ABB RobotStudio station: first_asignm.rspag

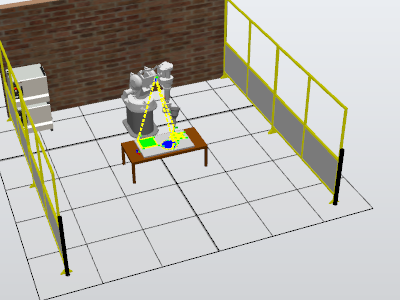
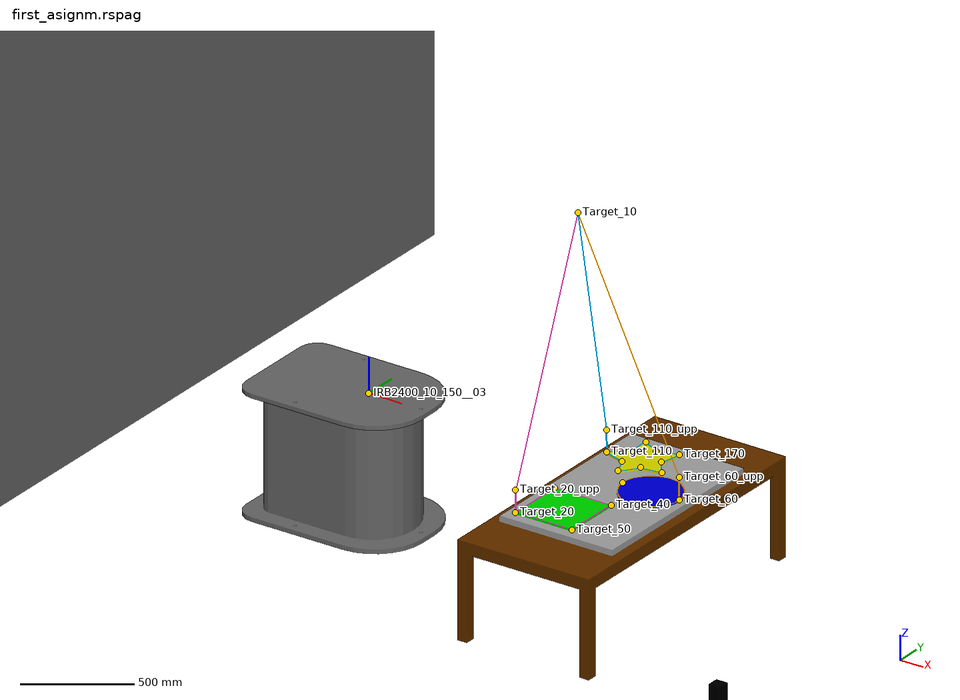
[picture v1: parts stored in the station drawn from their meshes, with robot base, taught points and paths (robot models come from the ABB library and are not in the file)]
--- station ---
Station first_asignm (saved by RobotStudio 24.1.10713.1)
Controller Controller2, task T_ROB1: task frame (RAPID world) sits at (2.56, -1.45, 620) mm, rotated rx 0 ry 0 rz -0.59 deg in the station
Controller Controller2
  mechanical unit ROB_1: IRB2400_10_150__03, 6 joints, base frame (0, 0, 0) mm
Layout (positions relative to the parent item):
  - IRB2400_10_150__03 [mechanism, from %ABB.RobotStudio.Models.IRB2400%\IRB2400_10_150_G_03.rslib] at (2.56, -1.45, 620) mm, rotated rx 0 ry 0 rz -0.59 deg; joint values [0.3771, 1.0223, 1.6235, 0.1721, -1.1317, 0.4182] (rad or m)
  - RobotStand2400H620 [part] at (0, 0, 0) mm, rotated rx 0 ry 0 rz -90 deg, size 600 x 830 x 620 mm
  - Table [part] at (1700, -750, 0) mm, rotated rx 0 ry 0 rz 90 deg, size 1500 x 700 x 488 mm
  - BackgroundWall [part] at (-1400, 2500, 0) mm, rotated rx 0 ry -90 rz 90 deg, size 2500 x 200 x 5000 mm
  - Fence_2500 [graphiccomponentgroup, from Equipment\Fence_2500.rslib] at (-1373.2, 2448.38, 0) mm, rotated rx 0 ry 0 rz -90 deg
    - Body 1 [part, from Equipment\Fence_2500.rslib]
    - Body 2 [part, from Equipment\Fence_2500.rslib]
  - Fence_2500_2 [graphiccomponentgroup, from Equipment\Fence_2500.rslib] at (1125.76, 2439.94, 0) mm, rotated rx 0 ry 0 rz -90 deg
    - Body 1 [part, from Equipment\Fence_2500.rslib]
    - Body 2 [part, from Equipment\Fence_2500.rslib]
  - Fence_2500_3 [graphiccomponentgroup, from Equipment\Fence_2500.rslib] at (-1386.44, -2458.41, 0) mm, rotated rx 0 ry 0 rz -90 deg
    - Body 1 [part, from Equipment\Fence_2500.rslib]
    - Body 2 [part, from Equipment\Fence_2500.rslib]
  - Fence_2500_4 [graphiccomponentgroup, from Equipment\Fence_2500.rslib] at (1081.61, -2474.76, 0) mm, rotated rx 0 ry 0 rz -90 deg
    - Body 1 [part, from Equipment\Fence_2500.rslib]
    - Body 2 [part, from Equipment\Fence_2500.rslib]
  - LightSensor [part] at (3608.83, 2403.41, 0) mm, size 60 x 60 x 1200 mm
  - LightSensor_2 [part] at (3563.84, -2499.97, 0) mm, size 60 x 60 x 1200 mm
  - supportframe2 [part] at (1050, 500, 488) mm, rotated rx 0 ry 0 rz -90 deg, size 1000 x 600 x 30 mm
  - star [part] at (1001.14, 175.39, 469.61) mm, rotated rx 0 ry 0 rz -18 deg, size 309.3 x 312.1 x 30 mm
  - cirkel [part] at (1023.03, -355.65, 518) mm, size 300 x 298.4 x 30 mm
  - kvadrat [part] at (460, -520, 516.18) mm, size 300 x 300 x 30 mm
  - gluetool [mechanism, from Assiment\gluetool.rslib] at (819.78, 298.44, 801.45) mm, rotated rx 143.42 ry 54.04 rz 148.38 deg
  - IRC5_Dual-Cabinet [part, from %ABB.RobotStudio.Models.IRC5%\IRC5_Dual-Cabinet.rslib] at (-784.69, -2074.47, 100) mm, rotated rx 90 ry 0 rz 90 deg
  - Part_2 [part] at (1023.03, -355.65, 518) mm, size 300 x 298.4 x 0 mm
Attachment: star is attached to supportframe2
Attachment: kvadrat is attached to supportframe2
Attachment: cirkel is attached to supportframe2
Attachment: supportframe2 is attached to Table
Attachment: gluetool is attached to IRB2400_10_150__03 / Link6

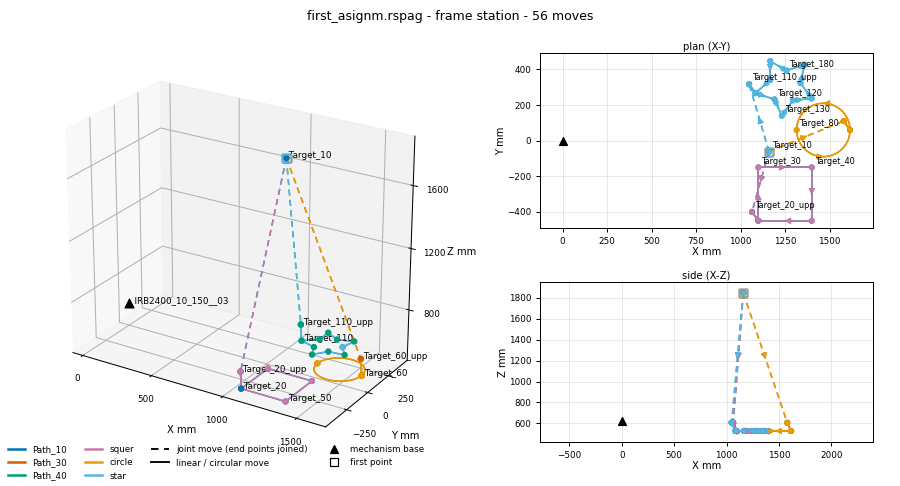
[picture p0: tool path of first_asignm.rspag in frame station, 56 of 56 moves have a stored position in this frame; points joined in program order, loops and branches not executed]
--- Backups/Controller2/RAPID/TASK1/PROGMOD/CalibData.mod ---
MODULE CalibData
    PERS tooldata gluetool:=[TRUE,[[47.792,-47.793,292.208],[0.923880453,0.270593988,0.27059897,0.000004062]],[1,[0,0,1],[1,0,0,0],0,0,0]];
    TASK PERS wobjdata Workobject_1:=[FALSE,TRUE,"",[[1465.9377766,-555.559495537,-110.643721572],[0.981995154,0.007735876,-0.020435156,0.187638159]],[[0,0,0],[1,0,0,0]]];
ENDMODULE

--- Backups/Controller2/RAPID/TASK1/PROGMOD/Module1.mod ---
MODULE Module1
        CONST robtarget Target_10:=[[-41.760657856,595.661836036,1334.239977499],[0.1634513,0.3686913,0.914955019,-0.014412176],[0,-1,0,0],[9E+09,9E+09,9E+09,9E+09,9E+09,9E+09]];
    CONST robtarget Target_20:=[[-293.739133821,244.320639444,27.648533238],[0.164058227,0.357731456,0.916814008,-0.067566099],[0,-1,0,0],[9E+09,9E+09,9E+09,9E+09,9E+09,9E+09]];
    CONST robtarget Target_30:=[[-186.145059876,524.28142208,20.904985353],[0.164039379,0.358304337,0.91678529,-0.064913921],[0,-1,0,0],[9E+09,9E+09,9E+09,9E+09,9E+09,9E+09]];
    CONST robtarget Target_40:=[[93.599135006,416.499861723,9.665738199],[0.163835348,0.362975372,0.916283469,-0.042795602],[0,-1,0,0],[9E+09,9E+09,9E+09,9E+09,9E+09,9E+09]];
    CONST robtarget Target_50:=[[-13.994938939,136.539079087,16.409286084],[0.164008319,0.359172644,0.916728515,-0.060869634],[0,-1,0,0],[9E+09,9E+09,9E+09,9E+09,9E+09,9E+09]];
    CONST robtarget Target_60:=[[369.476992779,535.242345722,-1.285956973],[0.164181139,0.345699668,0.915966091,-0.120591929],[0,-1,0,0],[9E+09,9E+09,9E+09,9E+09,9E+09,9E+09]];
    CONST robtarget Target_70:=[[283.40193231,729.113517218,0.961892661],[0.164180302,0.351853648,0.916729549,-0.094078551],[0,-1,0,0],[9E+09,9E+09,9E+09,9E+09,9E+09,9E+09]];
    CONST robtarget Target_80:=[[89.732797896,643.023906079,9.953290181],[0.164170715,0.352675827,0.916781174,-0.09044344],[0,-1,0,0],[9E+09,9E+09,9E+09,9E+09,9E+09,9E+09]];
    CONST robtarget Target_90:=[[175.807858365,449.152734583,7.705440546],[0.163487769,0.368236685,0.915092168,-0.016727716],[-1,-1,0,0],[9E+09,9E+09,9E+09,9E+09,9E+09,9E+09]];
    CONST robtarget Target_100:=[[369.476992779,535.242345722,-1.285956973],[0.164032525,0.338335776,0.914257142,-0.150851289],[0,-1,0,0],[9E+09,9E+09,9E+09,9E+09,9E+09,9E+09]];
    CONST robtarget Target_110:=[[-51.311674831,918.864864566,15.560999329],[0.164095805,0.356448324,0.916853669,-0.073460932],[0,-1,0,0],[9E+09,9E+09,9E+09,9E+09,9E+09,9E+09]];
    CONST robtarget Target_120:=[[35.611069333,848.29198306,12.348005726],[0.164181941,0.34578477,0.915980975,-0.120233261],[0,-1,0,0],[9E+09,9E+09,9E+09,9E+09,9E+09,9E+09]];
    CONST robtarget Target_130:=[[40.818568184,747.590756282,12.882109612],[0.164195884,0.348577196,0.916403541,-0.108342972],[0,-1,0,0],[9E+09,9E+09,9E+09,9E+09,9E+09,9E+09]];
    CONST robtarget Target_140:=[[129.808826796,805.323097391,8.613713401],[0.163772247,0.364097202,0.916087992,-0.037345285],[0,-1,0,0],[9E+09,9E+09,9E+09,9E+09,9E+09,9E+09]];
    CONST robtarget Target_150:=[[232.242262185,777.747137591,4.408706443],[0.164054081,0.357860896,0.916808121,-0.066967959],[0,-1,0,0],[9E+09,9E+09,9E+09,9E+09,9E+09,9E+09]];
    CONST robtarget Target_160:=[[204.856712118,880.316393149,4.815934456],[0.163731194,0.36477707,0.915954578,-0.034014637],[0,-1,0,0],[9E+09,9E+09,9E+09,9E+09,9E+09,9E+09]];
    CONST robtarget Target_170:=[[262.680463938,969.293462258,1.654828899],[0.163613768,0.366550779,0.91555164,-0.025224117],[0,-1,0,0],[9E+09,9E+09,9E+09,9E+09,9E+09,9E+09]];
    CONST robtarget Target_180:=[[156.76549339,974.952127682,6.174886911],[0.163831518,0.363046462,0.916271979,-0.042451873],[0,-1,0,0],[9E+09,9E+09,9E+09,9E+09,9E+09,9E+09]];
    CONST robtarget Target_190:=[[90.070200615,1057.517977687,8.426183116],[0.163939645,0.360848913,0.916572595,-0.052976713],[0,-1,0,0],[9E+09,9E+09,9E+09,9E+09,9E+09,9E+09]];
    CONST robtarget Target_200:=[[51.996100855,958.446029858,10.812529899],[0.163484758,0.368274734,0.915080909,-0.016534319],[0,-1,0,0],[9E+09,9E+09,9E+09,9E+09,9E+09,9E+09]];
    CONST robtarget Target_20_upp:=[[-305.599454825,304.750452419,106.436669969],[0.164055332,0.357822074,0.916809923,-0.067147424],[0,-1,0,0],[9E+09,9E+09,9E+09,9E+09,9E+09,9E+09]];
    CONST robtarget Target_60_upp:=[[357.616671775,595.672158697,77.502179758],[0.164166693,0.34443766,0.915731819,-0.125885782],[0,-1,0,0],[9E+09,9E+09,9E+09,9E+09,9E+09,9E+09]];
    CONST robtarget Target_110_upp:=[[-63.171995835,979.294677541,94.34913606],[0.16419453,0.347826437,0.916302665,-0.111563221],[0,-1,0,0],[9E+09,9E+09,9E+09,9E+09,9E+09,9E+09]];
!***********************************************************
    !
    ! Module:  Module1
    !
    ! Description:
    !   <Insert description here>
    !
    ! Author: haba0028
    !
    ! Version: 1.0
    !
    !***********************************************************


    !***********************************************************
    !
    ! Procedure main
    !
    !   This is the entry point of your program
    !
    !***********************************************************
    PROC main()
        !Add your code here
        Path_10;
        Path_30;
        Path_40;
        squer;
        circle;
        star;
    ENDPROC
    PROC Path_10()
        MoveJ Target_10,v1000,fine,gluetool\WObj:=Workobject_1;
        MoveJ Target_20_upp,v1000,fine,gluetool\WObj:=Workobject_1;
        MoveL Target_20,v1000,fine,gluetool\WObj:=Workobject_1;
        MoveL Target_30,v1000,fine,gluetool\WObj:=Workobject_1;
        MoveL Target_40,v1000,fine,gluetool\WObj:=Workobject_1;
        MoveL Target_50,v1000,fine,gluetool\WObj:=Workobject_1;
        MoveL Target_20,v1000,fine,gluetool\WObj:=Workobject_1;
        MoveJ Target_20_upp,v1000,fine,gluetool\WObj:=Workobject_1;
    ENDPROC
    PROC Path_30()
        MoveJ Target_10,v1000,fine,gluetool\WObj:=Workobject_1;
        MoveJ Target_60_upp,v1000,fine,gluetool\WObj:=Workobject_1;
        MoveL Target_60,v1000,fine,gluetool\WObj:=Workobject_1;
        MoveC Target_70,Target_80,v1000,fine,gluetool\WObj:=Workobject_1;
        MoveC Target_90,Target_100,v1000,fine,gluetool\WObj:=Workobject_1;
        MoveJ Target_60_upp,v1000,fine,gluetool\WObj:=Workobject_1;
    ENDPROC
    PROC Path_40()
        MoveJ Target_10,v1000,fine,gluetool\WObj:=Workobject_1;
        MoveJ Target_110_upp,v1000,fine,gluetool\WObj:=Workobject_1;
        MoveL Target_110,v1000,fine,gluetool\WObj:=Workobject_1;
        MoveL Target_120,v1000,fine,gluetool\WObj:=Workobject_1;
        MoveL Target_130,v1000,fine,gluetool\WObj:=Workobject_1;
        MoveL Target_140,v1000,fine,gluetool\WObj:=Workobject_1;
        MoveL Target_150,v1000,fine,gluetool\WObj:=Workobject_1;
        MoveL Target_160,v1000,fine,gluetool\WObj:=Workobject_1;
        MoveL Target_170,v1000,fine,gluetool\WObj:=Workobject_1;
        MoveL Target_180,v1000,fine,gluetool\WObj:=Workobject_1;
        MoveL Target_190,v1000,fine,gluetool\WObj:=Workobject_1;
        MoveL Target_200,v1000,fine,gluetool\WObj:=Workobject_1;
        MoveL Target_110,v1000,fine,gluetool\WObj:=Workobject_1;
        MoveJ Target_110_upp,v1000,fine,gluetool\WObj:=Workobject_1;
    ENDPROC
    PROC squer()
        MoveJ Target_10,v1000,fine,gluetool\WObj:=Workobject_1;
        MoveJ Target_20_upp,v1000,fine,gluetool\WObj:=Workobject_1;
        MoveL Target_20,v1000,fine,gluetool\WObj:=Workobject_1;
        MoveL Target_30,v1000,fine,gluetool\WObj:=Workobject_1;
        MoveL Target_40,v1000,fine,gluetool\WObj:=Workobject_1;
        MoveL Target_50,v1000,fine,gluetool\WObj:=Workobject_1;
        MoveL Target_20,v1000,fine,gluetool\WObj:=Workobject_1;
        MoveJ Target_20_upp,v1000,fine,gluetool\WObj:=Workobject_1;
    ENDPROC
    PROC circle()
        MoveJ Target_10,v1000,fine,gluetool\WObj:=Workobject_1;
        MoveJ Target_60_upp,v1000,fine,gluetool\WObj:=Workobject_1;
        MoveL Target_60,v1000,fine,gluetool\WObj:=Workobject_1;
        MoveC Target_70,Target_80,v1000,fine,gluetool\WObj:=Workobject_1;
        MoveC Target_90,Target_100,v1000,fine,gluetool\WObj:=Workobject_1;
        MoveJ Target_60_upp,v1000,fine,gluetool\WObj:=Workobject_1;
    ENDPROC
    PROC star()
        MoveJ Target_10,v1000,fine,gluetool\WObj:=Workobject_1;
        MoveJ Target_110_upp,v1000,fine,gluetool\WObj:=Workobject_1;
        MoveL Target_110,v1000,fine,gluetool\WObj:=Workobject_1;
        MoveL Target_120,v1000,fine,gluetool\WObj:=Workobject_1;
        MoveL Target_130,v1000,fine,gluetool\WObj:=Workobject_1;
        MoveL Target_140,v1000,fine,gluetool\WObj:=Workobject_1;
        MoveL Target_150,v1000,fine,gluetool\WObj:=Workobject_1;
        MoveL Target_160,v1000,fine,gluetool\WObj:=Workobject_1;
        MoveL Target_170,v1000,fine,gluetool\WObj:=Workobject_1;
        MoveL Target_180,v1000,fine,gluetool\WObj:=Workobject_1;
        MoveL Target_190,v1000,fine,gluetool\WObj:=Workobject_1;
        MoveL Target_200,v1000,fine,gluetool\WObj:=Workobject_1;
        MoveL Target_110,v1000,fine,gluetool\WObj:=Workobject_1;
        MoveJ Target_110_upp,v1000,fine,gluetool\WObj:=Workobject_1;
    ENDPROC
ENDMODULE
